(* CODESYS project do_fault_detect.20190114.1.project

Project tree, tasks and I/O mapping:
  Changsha_Xiangji_ARM_Cortex_A9_xilinx_zynq7000_linux : Changsha Xiangji-ARM Cortex A9(xilinx zynq7000)-linux, Changsha Xiangji Hiden Technology Co.Ltd, version 3.5.10.40
    application Application
      libraries: CAA Types Extern, 3.5.10.0 (CAA Technical Workgroup); VisuDialogs, * (System); CAA Real Time Clock Extern, 3.5.10.0 (CAA Technical Workgroup); CAA Callback Extern, 3.5.11.0 (CAA Technical Workgroup); CAA Can Low Level Extern, 3.5.11.0 (CAA Technical Workgroup); CAA Can Low Level Imp Extern, 3.5.11.0 (CAA Technical Workgroup); SysMem, 3.5.12.0 (System); CAA Net Base Services, 3.5.12.0 (CAA Technical Workgroup); Standard, 3.5.12.0 (System); CAA SerialCom, 3.5.12.0 (CAA Technical Workgroup); CAA File, 3.5.12.0 (CAA Technical Workgroup); CAA DTUtil Extern, 3.5.12.0 (CAA Technical Workgroup)
      task Task (cyclic, interval 50 ms, priority 1) calls prg_main
      program prg_main [ST]
      FBs/
        function block FB_DOH_FAULT [ST]
    SoftMotion General Axis Pool
    IoDrvMIC7001 : IoDrvMIC7001, Cyber-MI, version 18.11.1
        input  Application.prg_main.ai_18 : DWORD  // Ai18-Do00@C25
        input  Application.prg_main.ai_23 : DWORD  // Ai23-Do05@C04
        output Application.prg_main.do_00 : BOOL  // Do00-Ai18@C25
        output Application.prg_main.do_05 : BOOL  // Do05-Ai23@C04
        unmapped channels: Ai00@C16, Ai01@C28, Ai02@C17, Ai03@C29, Ai04@C30, Ai05@C19, Ai06@C31, Ai07@C20, Ai08@C18, Ai09@D18, Ai10@D20, Ai11@D31, Ai12@D19, Ai13@D30, Ai14@D29, Ai15@D17, Ai16@D28, Ai17@D16, Ai19-Do01@C24, Ai20-Do02@C13, Ai21-Do03@C01, Ai22-Do04@C03, Ai24-Do06@C05, Ai25-Do07@C06, Ai26-Do08@C08, Ai27-Do09@C09, Ai28-Do10@C10, Ai29-Do11@C11, Ai30-Do12@D34, Ai31-Do13@D35, Ai32-Do14@D23, Ai33-Do15@D12, Ai34-Do16@D10, Ai35-Do17@D09, Ai36-Do18@D08, Ai37-Do19@D07, Ai38-Do20@D05, Ai39-Do21@D04, Ai40-Do22@D03, Ai41-Do23@D02,
          Ai42-Do24@C23, Ai43-Do25@C35, Ai44-Do26@D24, Ai45-Do27@D13, Ai46-Ao00@C22, Ai47-Ao01@D14, Ai48_Pi02, Ai49_Out5V, Ai50_VCC, Ai51_VCC_L, Ai52_VCC_R, Ai53_Pwm-i0, Ai54_Pwm-i1, Ai55_Pwm-i2, Ai56_Pwm-i3, Ai57_CPU-T, Ai58_G-x, Ai59_G-y, Ai60_G-z, Ai61-reserved, Ai62-IO-cntr, Ai63-CDS-cntr, Di00-Ai00@C16, Di01-Ai01@C28, Di02-Ai02@C17, Di03-Ai03@C29, Di04-Ai04@C30, Di05-Ai05@C19, Di06-Ai06@C31, Di07-Ai07@C20, Di08-Ai08@C18, Di09-Ai09@D18, Di10-Ai10@D20, Di11-Ai11@D31, Di12-Ai12@D19, Di13-Ai13@D30, Di14-Ai14@D29, Di15-Ai15@D17, Di16-Ai16@D28, Di17-Ai17@D16,
          Di18-Ai18@C25, Di19-Ai19@C24, Di20-Ai20@C13, Di21-Ai21@C01, Di22-Ai22@C03, Di23-Ai23@C04, Di24-Ai24@C05, Di25-Ai25@C06, Di26-Ai26@C08, Di27-Ai27@C09, Di28-Ai28@C10, Di29-Ai29@C11, Di30-Ai30@D34, Di31-Ai31@D35, Di32-Ai32@D23, Di33-Ai33@D12, Di34-Ai34@D10, Di35-Ai35@D09, Di36-Ai36@D08, Di37-Ai37@D07, Di38-Ai38@D05, Di39-Ai39@D04, Di40-Ai40@D03, Di41-Ai41@D02, Di42-Ai42@C23, Di43-Ai43@C35, Di44-Ai44@D24, Di45-Ai45@D13, Di46-Ai46@C22, Di47-Ai47@D14, Di48-Pi00@C15, Di49-Pi01@C14, Di50-Pi02@D22, Di51-Pi03@D21, Di52-reserved, Di53-reserved, Di54-reserved, Di55-reserved, Di56-reserved, Di57-reserved,
          Di58-reserved, Di59-reserved, Di60-reserved, Di61-reserved, Di62-reserved, Di63-reserved, Pi00-Di48@C15, Pi01-Di49@C14, Pi02-Di50@D22, Pi03-Di51@D21, Do01-Ai19@C24, Do02-Ai20@C13, Do03-Ai21@C01, Do04-Ai22@C03, Do06-Ai24@C05, Do07-Ai25@C06, Do08-Ai26@C08, Do09-Ai27@C09, Do10-Ai28@C10, Do11-Ai29@C11, Do12-Ai30@D34, Do13-Ai31@D35, Do14-Ai32@D23, Do15-Ai33@D12, Do16-Ai34@D10, Do17-Ai35@D09, Do18-Ai36@D08, Do19-Ai37@D07, Do20-Ai38@D05, Do21-Ai39@D04, Do22-Ai40@D03, Do23-Ai41@D02, Do24-Ai42@C23, Do25-Ai43@C35, Do26-Ai44@D24, Do27-Ai45@D13, Do28-Pwmi00@C33, Do29-Pwmi01@C34, Do30-Pwmi02@D25, Do31-Pwmi03@D26,
          PWM00@C25, PWM01@C24, PWM02@C13, PWM03@C01, PWM04@C03, PWM05@C04, PWM06@C05, PWM07@C06, PWM08@C08, PWM09@C09, PWM10@C10, PWM11@C11, PWM12@D34, PWM13@D35, PWM14@D23, PWM15@D12, PWM16@D10, PWM17@D09, PWM18@D08, PWM19@D07, PWM20@D05, PWM21@D04, PWM22@D03, PWM23@D02, PWM24@C23, PWM25@C35, PWM26@D24, PWM27@D13, PWM28-Pwmi00@C33, PWM29-Pwmi01@C34, PWM30-Pwmi02@D25, PWM31-Pwmi03@D26, PWM_I_0@C33, PWM_I_1@C34, PWM_I_2@D25, PWM_I_3@D26, Ao00-Ai46@C22, Ao01-Ai47@D14, LED_run, LED_err,
          LED_usr, ctrl_ai_raw, ctrl_adjust, ctrl_adj0, ctrl_adj1, ctrl_adj2, ctrl_adj3, ctrl_adj4
  5ce3da45-db07-42e7-a21c-a00fff4ed8f6|C:\Users\Administrator\Desktop\robotview1.bmp
  5ce3da45-db07-42e7-a21c-a00fff4ed8f6|C:\Users\Administrator\Desktop\robotview2.bmp
  text list GlobalTextList
  5ce3da45-db07-42e7-a21c-a00fff4ed8f6|C:\Users\Administrator\Desktop\1129.bmp
  5ce3da45-db07-42e7-a21c-a00fff4ed8f6|C:\Users\Administrator\Desktop\robotview0.bmp
*)

// Changsha_Xiangji_ARM_Cortex_A9_xilinx_zynq7000_linux/Application/prg_main
PROGRAM prg_main
VAR
	do_00:BOOL;  //do-00, 需绑定到对应的IO端口
	ai_18:DWORD; //ai-18, 需绑定到对应的IO端口
	
	do_fault_00 :FB_DOH_FAULT;  //创建故障诊断功能块的实例，每个DO端口创建一个
	do_01_short_flag :BOOL := FALSE;  //短路标志
	do_01_open_flag :BOOL := FALSE;   //开路标志	

(**************************************************************************)

	do_05:BOOL;  //do-00, 需绑定到对应的IO端口
	ai_23:DWORD; //ai-18, 需绑定到对应的IO端口
	
	do_fault_05 :FB_DOH_FAULT;  //创建故障诊断功能块的实例，每个DO端口创建一个	
	
	do_05_short_flag :BOOL := FALSE;  //短路标志
	do_05_open_flag :BOOL := FALSE;   //开路标志
END_VAR


do_fault_00(enable := TRUE,dout := do_00, ai := ai_18);
do_01_short_flag := do_fault_00.short;
do_01_open_flag := do_fault_00.open;


do_fault_05(enable := TRUE, dout := do_05, ai := ai_23);
do_05_short_flag := do_fault_05.short;
do_05_open_flag := do_fault_05.open;

RETURN;

END_PROGRAM

// Changsha_Xiangji_ARM_Cortex_A9_xilinx_zynq7000_linux/Application/FBs/FB_DOH_FAULT
FUNCTION_BLOCK FB_DOH_FAULT      //检测MIC7000系列控制器高有效输出端口的短路和短线故障 功能块
VAR_INPUT
	enable :BOOL;   //开关，true 表示启用本功能块
	dout:BOOL;     	//需要检测的高有效开关量输出端口值
	ai:DWORD;      	//需要检测的高有效输出端口对应的模拟量输入值
END_VAR
VAR_OUTPUT
	ok:BOOL;    	//正常标志，为true表示无故障
	short:BOOL;  	//短路故障标志
	open:BOOL;    	//短线故障标志
END_VAR

VAR
	stat: DWORD := 0;
	stat_short :DWORD := 0;
	stat_open :DWORD := 0;
	short_cntr :DWORD := 0;
	open_cntr :DWORD := 0;
END_VAR

VAR CONSTANT   //参数定义，可以根据情况修改
	SHORT_VALUE :DWORD := 3000; //短路门槛值
	OPEN_VALUE :DWORD := 25;   	//开路门槛值
	TIME_OUT :DWORD := 10;   	//超时周期数
END_VAR

IF NOT enable THEN
	ok := TRUE;
	short := FALSE;
	open := FALSE;
	short_cntr := 0;
	open_cntr := 0;
	RETURN;
END_IF

CASE stat OF
	0:
		ok := TRUE;
		short := FALSE;
		open := FALSE;
		IF dout THEN  
			stat := 100;	// dout high, detect short
			stat_short := 0;
		ELSE 
			stat := 200;  //dout low, detect open
			stat_open := 0;
		END_IF
	
	100:  //detect short
		IF NOT dout THEN  //return 
			stat := 0;
		END_IF
		CASE stat_short OF
			0:
				short := FALSE;
				IF ai < SHORT_VALUE THEN  //short
					stat_short := 10;
					short_cntr := 0;
				END_IF
			10:  //short wait for timeout
				IF ai > SHORT_VALUE THEN  //normal , wait for return
					IF short_cntr = 0 THEN
						stat_short := 0;
					ELSE
						short_cntr := short_cntr - 1;
					END_IF
				ELSE  //short, 
					IF short_cntr > TIME_OUT THEN
						short := TRUE;
					ELSE
						short_cntr := short_cntr + 1;
					END_IF		
				END_IF	
		END_CASE

	200:
		IF dout THEN  //  dout high, return to detect short
			stat := 0;
		END_IF
		CASE stat_open OF
			0:
				open := FALSE;
				IF ai > OPEN_VALUE THEN  //open
					stat_open := 10;
					open_cntr := 0;
				END_IF
			10:
				IF ai < OPEN_VALUE THEN  //normal, wait for return
					IF open_cntr = 0 THEN
						stat_open := 0;
					ELSE
						open_cntr := open_cntr - 1;
					END_IF
				ELSE
					IF open_cntr > TIME_OUT THEN
						open := TRUE;
					ELSE
						open_cntr := open_cntr + 1;
					END_IF
				END_IF			
		END_CASE
END_CASE

ok := (NOT short) AND (NOT open);

END_FUNCTION_BLOCK
